# EPICS autosave request: iocBoot/iocScreen/auto_settings_screen.req
file screen.req       P=$(P), R=$(R)
